// TIA Portal V20 export
// export: Created 2025-12-01T14:57:26.4482814Z, ExportSetting None, DisplayName Totally Integrated Automation Portal, DisplayVersion V20 Update 3, DisplayName TIA Portal Openness, DisplayVersion V20 Update 3, DisplayName TIA Portal Version Control Interface, DisplayVersion V20 Update 3, DisplayName STEP 7 Professional, DisplayVersion V20 Update 3, DisplayName STEP 7 Safety, DisplayVersion V20 Update 2, DisplayName WinCC Basic/Comfort/Advanced, DisplayVersion V20 Update 3, DisplayName WinCC Professional, DisplayVersion V20 Update 3, DisplayName WinCC Unified, DisplayVersion V20 Update 3
DATA_BLOCK "DB601_PeinesQuimarox"   // DB601
{ S7_Optimized_Access := 'FALSE' }
AUTHOR : Naibes
// stored: AutoNumber false
   VAR RETAIN
      Quimarox : Array[1.."CTE_MaxNumQuimarox"] of Struct
         vagon { S7_SetPoint := 'True'} : Array[1.."CTE_MaxNumVagones"] of "CBS_Carrier";
      END_STRUCT;
   END_VAR
BEGIN
END_DATA_BLOCK
